// TIA Portal V19 export
VAR_GLOBAL   // PLC tag table "LB212"
   LB212_Carriage_Lp_BWD AT %Q121.2 : Bool;   // 339SH2
   LB212_Carriage_Lp_FWD AT %Q121.1 : Bool;   // 339SH1
   LB212_Carriage_Pb_BWD AT %I124.6 : Bool;   // 339SH2
   LB212_Carriage_Pb_FWD AT %I124.5 : Bool;   // 339SH1
   LB212_DieClamp_Lp_Rest AT %Q120.2 : Bool;   // 338HL2
   LB212_DieClamp_Lp_Work AT %Q120.1 : Bool;   // 338HL1
   LB212_DieClamp_Pb_Rest AT %I123.6 : Bool;   // 338SH2
   LB212_DieClamp_Pb_Work AT %I123.5 : Bool;   // 338SH1
   LB212_DieSetOP_Lp_Req AT %Q120.0 : Bool;   // 338HL1
   LB212_DiesOP_T1_Lp_Rest AT %Q120.3 : Bool;   // 338HL3
   LB212_DiesOP_T1_Lp_Work AT %Q120.4 : Bool;   // 338HL4
   LB212_DiesOP_T1_Pb_Rest AT %I123.7 : Bool;   // 338SH3
   LB212_DiesOP_T1_Pb_Work AT %I124.0 : Bool;   // 338SH4
   LB212_DiesOP_T2_Lp_Rest AT %Q120.5 : Bool;   // 388 - LIBERO
   LB212_DiesOP_T2_Lp_Work AT %Q120.6 : Bool;   // 388 - LIBERO
   LB212_DiesOP_T3_Lp_Rest AT %Q120.7 : Bool;   // 388 - LIBERO
   LB212_DiesOP_T3_Lp_Work AT %Q121.0 : Bool;   // 388 - LIBERO
   LB212_RollFormer_Lp_BWD AT %Q121.4 : Bool;   // 339SH3
   LB212_RollFormer_Lp_FWD AT %Q121.3 : Bool;   // 339SH4
   LB212_RollFormer_Pb_BWD AT %I125.0 : Bool;   // 339SH4
   LB212_RollFormer_Pb_FWD AT %I124.7 : Bool;   // 339SH3
   LB212_Button_L AT %I1079.3 : Bool;   // 106DI3 - 244SB1
   LB212_Button_R AT %I1079.7 : Bool;   // 106DI7 - 244SB2
   LB212_DiesOP_T3_Pb_Rest AT %I124.3 : Bool;   // 388 - LIBERO
   LB212_DiesOP_T3_Pb_Work AT %I124.4 : Bool;   // 388 - LIBERO
   LB212_DiesOP_T2_Pb_Rest AT %I124.1 : Bool;   // 388 - LIBERO
   LB212_DiesOP_T2_Pb_Work AT %I124.2 : Bool;   // 388 - LIBERO
END_VAR
